(* CODESYS project Flight Simulator.project
   CompiledLibraryCompatibilityVersion: CODESYS V3.5 SP16 Patch 7

Project tree, tasks and I/O mapping:
  PLC : HX-CP1S08, Hitachi Industrial Equipment Systems Co., Ltd., order no. HX-CP1S08, version 3.5.8.24
      settings: IP Address = '192.168.137.20'
    application Application
      libraries: Unit Conversion Interfaces, * (Intern); Standard, * (System); VisuDialogs, * (System); CAA Device Diagnosis, 3.5.4.0 (CAA Technical Workgroup); CAA Net Base Services, 3.5.8.10 (CAA Technical Workgroup); NetVarUdp, 3.5.17.0 (System); PRO JSON, 1.0.0.13 (Pro Electric)
      task EtherCAT_Task (cyclic, interval 8 ms, priority 1) calls nothing
      task VISU_TASK (cyclic, interval 200 ms, priority 31) calls VisuElems.Visu_Prg
      task Task (cyclic, interval 5 ms, priority 1) calls main, TcpClient
      global variables gvlSetting
      data type ServoData
      program TcpClient [ST]
      program main [ST]
      visualisation Main
      global variables GVL
    SoftMotion General Axis Pool : SoftMotion General Axis Pool, 3S - Smart Software Solutions GmbH, version 4.9.0.0
      SM_Drive_Virtual : SM_Drive_Virtual, 3S - Smart Software Solutions GmbH, order no. 1805, version 4.0.0.0
          settings: wDriveID = 6
    Basic : Basic, Hitachi-IES, version 3.5.8.20
      _16_Digital_Input : 16 Digital Input, Hitachi-IES, version 3.4.0.0
          input  Application.GVL.resetButton : BOOL  // ReserveWord0Type.Bit1
          input  Application.GVL.startButton : BOOL  // ReserveWord0Type.Bit2
          input  Application.GVL.stopButton : BOOL  // ReserveWord0Type.Bit3
          input  Application.GVL.safetySystem : BOOL  // ReserveWord0Type.Bit4
          unmapped channels: ReserveWord0Type, ReserveWord0Type, ReserveWord0Type
      _16_Digital_Output : 16 Digital Output, Hitachi-IES, version 3.4.0.0
          output Application.GVL.LightGreen : BOOL  // ReserveWord0Type.Bit0
          output Application.GVL.LightYellow : BOOL  // ReserveWord0Type.Bit1
          output Application.GVL.LightRed : BOOL  // ReserveWord0Type.Bit2
          unmapped channels: ReserveWord0Type, ReserveWord0Type, ReserveWord0Type
      <Empty>
      <Empty>
      _16_Digital_Input_1 : 16 Digital Input, Hitachi-IES, version 3.4.0.0
          unmapped channels: ReserveWord0Type, ReserveWord0Type, ReserveWord0Type
      <Empty>
      <Empty>
      <Empty>
      <Empty>
      <Empty>
      _16_Digital_Output_1 : 16 Digital Output, Hitachi-IES, version 3.4.0.0
          unmapped channels: ReserveWord0Type, ReserveWord0Type, ReserveWord0Type
    EtherCAT_Master : EtherCAT Master, Festo, version 3.5.16.43
        settings: MasterUseLRW = False; SlaveAutoRestart = True; NetworkName = 'eth2'; NetworkName = "eth2"; SelectNetworkByName = False; EnableTaskMessage = False; SrcAddress1 = 42135; SrcAddress2 = 3137775364; EnableSecondAdapter = False; SrcAddress = [16#A4,16#97,16#BB,16#06,16#A7,16#04]; NetworkName = 'eth2'; NetworkName = "eth2"; SelectNetworkByName = False
      servo_drive_2 : CMMT-AS (SoftMotion), Festo, order no. 5340819, 5340820, version 4.0.20.0
          settings: StationAlias = 0; Number of SDO = 1; Modes of operation.Index = 16#6060; Modes of operation.Subindex = 16#00; Modes of operation.Value = 8; Modes of operation.Size = 8; Modes of operation.AbortIfError = FALSE; Modes of operation.JumpToLine = FALSE; Modes of operation.Line = 0; Modes of operation.CompleteAccess = False
          unmapped channels: Controlword, Modes of operation, Target position, Profile velocity, Target velocity, Target torque, Velocity offset, Torque offset, Touch probe function, ---, Statusword, Modes of operation display, Position actual value, Velocity actual value, Torque actual value, Touch probe status, Touch probe 1 positive edge, Touch probe 1 negative edge, Touch probe 2 positive edge, Touch probe 2 negative edge, ---
        SM_Drive_EtherCAT_Festo_CMMT_AS_1 : SM_Drive_EtherCAT_Festo_CMMT_AS, Festo, version 4.0.20.0
            settings: AdrOffset_8010 = 36; BitOffset_8010 = 0; BitLength_8010 = 16; Address_8010 = '%QW18'; Type_8010 = 'UINT'; AddressPointer_8010 = ADR(%QW18); AdrOffset_8020 = 38; BitOffset_8020 = 0; BitLength_8020 = 8; Address_8020 = '%QB38'; Type_8020 = 'SINT'; AddressPointer_8020 = ADR(%QB38); AdrOffset_8030 = 40; BitOffset_8030 = 0; BitLength_8030 = 32; Address_8030 = '%QD10'; Type_8030 = 'DINT'; AddressPointer_8030 = ADR(%QD10); AdrOffset_8040 = 48; BitOffset_8040 = 0; BitLength_8040 = 32; Address_8040 = '%QD12'; Type_8040 = 'DINT'; AddressPointer_8040 = ADR(%QD12); AdrOffset_8050 = 52; BitOffset_8050 = 0; BitLength_8050 = 16; Address_8050 = '%QW26'; Type_8050 = 'INT'; AddressPointer_8050 = ADR(%QW26); AdrOffset_8060 = 62; BitOffset_8060 = 0; BitLength_8060 = 16; Address_8060 = '%QW31'; Type_8060 = 'UINT'; AddressPointer_8060 = ADR(%QW31); AdrOffset_8510 = 40; BitOffset_8510 = 0; BitLength_8510 = 16; Address_8510 = '%IW20';
              Type_8510 = 'UINT'; AddressPointer_8510 = ADR(%IW20); AdrOffset_8520 = 42; BitOffset_8520 = 0; BitLength_8520 = 8; Address_8520 = '%IB42'; Type_8520 = 'SINT'; AddressPointer_8520 = ADR(%IB42); AdrOffset_8530 = 44; BitOffset_8530 = 0; BitLength_8530 = 32; Address_8530 = '%ID11'; Type_8530 = 'DINT'; AddressPointer_8530 = ADR(%ID11); AdrOffset_8540 = 48; BitOffset_8540 = 0; BitLength_8540 = 32; Address_8540 = '%ID12'; Type_8540 = 'DINT'; AddressPointer_8540 = ADR(%ID12); AdrOffset_8550 = 52; BitOffset_8550 = 0; BitLength_8550 = 16; Address_8550 = '%IW26'; Type_8550 = 'INT'; AddressPointer_8550 = ADR(%IW26); AdrOffset_8560 = 54; BitOffset_8560 = 0; BitLength_8560 = 16; Address_8560 = '%IW27'; Type_8560 = 'UINT'; AddressPointer_8560 = ADR(%IW27); AdrOffset_8570 = 56; BitOffset_8570 = 0; BitLength_8570 = 32; Address_8570 = '%ID14'; Type_8570 = 'DINT'; AddressPointer_8570 = ADR(%ID14); AdrOffset_8580 = 60; BitOffset_8580 = 0;
              BitLength_8580 = 32; Address_8580 = '%ID15'; Type_8580 = 'DINT'; AddressPointer_8580 = ADR(%ID15); AdrOffset_8590 = 64; BitOffset_8590 = 0; BitLength_8590 = 32; Address_8590 = '%ID16'; Type_8590 = 'DINT'; AddressPointer_8590 = ADR(%ID16); AdrOffset_8600 = 68; BitOffset_8600 = 0; BitLength_8600 = 32; Address_8600 = '%ID17'; Type_8600 = 'DINT'; AddressPointer_8600 = ADR(%ID17)
      servo_drive_1 : CMMT-AS (SoftMotion), Festo, order no. 5340819, 5340820, version 4.0.20.0
          settings: StationAlias = 0; Number of SDO = 1; Modes of operation.Index = 16#6060; Modes of operation.Subindex = 16#00; Modes of operation.Value = 8; Modes of operation.Size = 8; Modes of operation.AbortIfError = FALSE; Modes of operation.JumpToLine = FALSE; Modes of operation.Line = 0; Modes of operation.CompleteAccess = False
          unmapped channels: Controlword, Modes of operation, Target position, Profile velocity, Target velocity, Target torque, Velocity offset, Torque offset, Touch probe function, ---, Statusword, Modes of operation display, Position actual value, Velocity actual value, Torque actual value, Touch probe status, Touch probe 1 positive edge, Touch probe 1 negative edge, Touch probe 2 positive edge, Touch probe 2 negative edge, ---
        SM_Drive_EtherCAT_Festo_CMMT_AS : SM_Drive_EtherCAT_Festo_CMMT_AS, Festo, version 4.0.20.0
            settings: wDriveID = 0; AdrOffset_8010 = 4; BitOffset_8010 = 0; BitLength_8010 = 16; Address_8010 = '%QW2'; Type_8010 = 'UINT'; AddressPointer_8010 = ADR(%QW2); AdrOffset_8020 = 6; BitOffset_8020 = 0; BitLength_8020 = 8; Address_8020 = '%QB6'; Type_8020 = 'SINT'; AddressPointer_8020 = ADR(%QB6); AdrOffset_8030 = 8; BitOffset_8030 = 0; BitLength_8030 = 32; Address_8030 = '%QD2'; Type_8030 = 'DINT'; AddressPointer_8030 = ADR(%QD2); AdrOffset_8040 = 16; BitOffset_8040 = 0; BitLength_8040 = 32; Address_8040 = '%QD4'; Type_8040 = 'DINT'; AddressPointer_8040 = ADR(%QD4); AdrOffset_8050 = 20; BitOffset_8050 = 0; BitLength_8050 = 16; Address_8050 = '%QW10'; Type_8050 = 'INT'; AddressPointer_8050 = ADR(%QW10); AdrOffset_8060 = 30; BitOffset_8060 = 0; BitLength_8060 = 16; Address_8060 = '%QW15'; Type_8060 = 'UINT'; AddressPointer_8060 = ADR(%QW15); AdrOffset_8510 = 4; BitOffset_8510 = 0; BitLength_8510 = 16;
              Address_8510 = '%IW2'; Type_8510 = 'UINT'; AddressPointer_8510 = ADR(%IW2); AdrOffset_8520 = 6; BitOffset_8520 = 0; BitLength_8520 = 8; Address_8520 = '%IB6'; Type_8520 = 'SINT'; AddressPointer_8520 = ADR(%IB6); AdrOffset_8530 = 8; BitOffset_8530 = 0; BitLength_8530 = 32; Address_8530 = '%ID2'; Type_8530 = 'DINT'; AddressPointer_8530 = ADR(%ID2); AdrOffset_8540 = 12; BitOffset_8540 = 0; BitLength_8540 = 32; Address_8540 = '%ID3'; Type_8540 = 'DINT'; AddressPointer_8540 = ADR(%ID3); AdrOffset_8550 = 16; BitOffset_8550 = 0; BitLength_8550 = 16; Address_8550 = '%IW8'; Type_8550 = 'INT'; AddressPointer_8550 = ADR(%IW8); AdrOffset_8560 = 18; BitOffset_8560 = 0; BitLength_8560 = 16; Address_8560 = '%IW9'; Type_8560 = 'UINT'; AddressPointer_8560 = ADR(%IW9); AdrOffset_8570 = 20; BitOffset_8570 = 0; BitLength_8570 = 32; Address_8570 = '%ID5'; Type_8570 = 'DINT'; AddressPointer_8570 = ADR(%ID5); AdrOffset_8580 = 24;
              BitOffset_8580 = 0; BitLength_8580 = 32; Address_8580 = '%ID6'; Type_8580 = 'DINT'; AddressPointer_8580 = ADR(%ID6); AdrOffset_8590 = 28; BitOffset_8590 = 0; BitLength_8590 = 32; Address_8590 = '%ID7'; Type_8590 = 'DINT'; AddressPointer_8590 = ADR(%ID7); AdrOffset_8600 = 32; BitOffset_8600 = 0; BitLength_8600 = 32; Address_8600 = '%ID8'; Type_8600 = 'DINT'; AddressPointer_8600 = ADR(%ID8)
      servo_drive_3 : CMMT-AS (SoftMotion), Festo, order no. 5340819, 5340820, version 4.0.22.0
          settings: StationAlias = 0; Number of SDO = 1; Modes of operation.Index = 16#6060; Modes of operation.Subindex = 16#00; Modes of operation.Value = 8; Modes of operation.Size = 8; Modes of operation.AbortIfError = FALSE; Modes of operation.JumpToLine = FALSE; Modes of operation.Line = 0; Modes of operation.CompleteAccess = False
          unmapped channels: Controlword, Modes of operation, Target position, Profile velocity, Target velocity, Target torque, Velocity offset, Torque offset, Touch probe function, ---, Statusword, Modes of operation display, Position actual value, Velocity actual value, Torque actual value, Touch probe status, Touch probe 1 positive edge, Touch probe 1 negative edge, Touch probe 2 positive edge, Touch probe 2 negative edge, ---
        SM_Drive_EtherCAT_Festo_CMMT_AS_2 : SM_Drive_EtherCAT_Festo_CMMT_AS, Festo, version 4.0.22.0
            settings: wDriveID = 2; AdrOffset_8010 = 68; BitOffset_8010 = 0; BitLength_8010 = 16; Address_8010 = '%QW34'; Type_8010 = 'UINT'; AddressPointer_8010 = ADR(%QW34); AdrOffset_8020 = 70; BitOffset_8020 = 0; BitLength_8020 = 8; Address_8020 = '%QB70'; Type_8020 = 'SINT'; AddressPointer_8020 = ADR(%QB70); AdrOffset_8030 = 72; BitOffset_8030 = 0; BitLength_8030 = 32; Address_8030 = '%QD18'; Type_8030 = 'DINT'; AddressPointer_8030 = ADR(%QD18); AdrOffset_8040 = 80; BitOffset_8040 = 0; BitLength_8040 = 32; Address_8040 = '%QD20'; Type_8040 = 'DINT'; AddressPointer_8040 = ADR(%QD20); AdrOffset_8050 = 84; BitOffset_8050 = 0; BitLength_8050 = 16; Address_8050 = '%QW42'; Type_8050 = 'INT'; AddressPointer_8050 = ADR(%QW42); AdrOffset_8060 = 94; BitOffset_8060 = 0; BitLength_8060 = 16; Address_8060 = '%QW47'; Type_8060 = 'UINT'; AddressPointer_8060 = ADR(%QW47); AdrOffset_8510 = 76; BitOffset_8510 = 0; BitLength_8510 = 16;
              Address_8510 = '%IW38'; Type_8510 = 'UINT'; AddressPointer_8510 = ADR(%IW38); AdrOffset_8520 = 78; BitOffset_8520 = 0; BitLength_8520 = 8; Address_8520 = '%IB78'; Type_8520 = 'SINT'; AddressPointer_8520 = ADR(%IB78); AdrOffset_8530 = 80; BitOffset_8530 = 0; BitLength_8530 = 32; Address_8530 = '%ID20'; Type_8530 = 'DINT'; AddressPointer_8530 = ADR(%ID20); AdrOffset_8540 = 84; BitOffset_8540 = 0; BitLength_8540 = 32; Address_8540 = '%ID21'; Type_8540 = 'DINT'; AddressPointer_8540 = ADR(%ID21); AdrOffset_8550 = 88; BitOffset_8550 = 0; BitLength_8550 = 16; Address_8550 = '%IW44'; Type_8550 = 'INT'; AddressPointer_8550 = ADR(%IW44); AdrOffset_8560 = 90; BitOffset_8560 = 0; BitLength_8560 = 16; Address_8560 = '%IW45'; Type_8560 = 'UINT'; AddressPointer_8560 = ADR(%IW45); AdrOffset_8570 = 92; BitOffset_8570 = 0; BitLength_8570 = 32; Address_8570 = '%ID23'; Type_8570 = 'DINT'; AddressPointer_8570 = ADR(%ID23); AdrOffset_8580 = 96;
              BitOffset_8580 = 0; BitLength_8580 = 32; Address_8580 = '%ID24'; Type_8580 = 'DINT'; AddressPointer_8580 = ADR(%ID24); AdrOffset_8590 = 100; BitOffset_8590 = 0; BitLength_8590 = 32; Address_8590 = '%ID25'; Type_8590 = 'DINT'; AddressPointer_8590 = ADR(%ID25); AdrOffset_8600 = 104; BitOffset_8600 = 0; BitLength_8600 = 32; Address_8600 = '%ID26'; Type_8600 = 'DINT'; AddressPointer_8600 = ADR(%ID26)
      servo_drive_4 : CMMT-AS (SoftMotion), Festo, order no. 5340819, 5340820, version 4.0.20.0
          settings: StationAlias = 0; Number of SDO = 1; Modes of operation.Index = 16#6060; Modes of operation.Subindex = 16#00; Modes of operation.Value = 8; Modes of operation.Size = 8; Modes of operation.AbortIfError = FALSE; Modes of operation.JumpToLine = FALSE; Modes of operation.Line = 0; Modes of operation.CompleteAccess = False
          unmapped channels: Controlword, Modes of operation, Target position, Profile velocity, Target velocity, Target torque, Velocity offset, Torque offset, Touch probe function, ---, Statusword, Modes of operation display, Position actual value, Velocity actual value, Torque actual value, Touch probe status, Touch probe 1 positive edge, Touch probe 1 negative edge, Touch probe 2 positive edge, Touch probe 2 negative edge, ---
        SM_Drive_EtherCAT_Festo_CMMT_AS_3 : SM_Drive_EtherCAT_Festo_CMMT_AS, Festo, version 4.0.20.0
            settings: wDriveID = 3; AdrOffset_8010 = 100; BitOffset_8010 = 0; BitLength_8010 = 16; Address_8010 = '%QW50'; Type_8010 = 'UINT'; AddressPointer_8010 = ADR(%QW50); AdrOffset_8020 = 102; BitOffset_8020 = 0; BitLength_8020 = 8; Address_8020 = '%QB102'; Type_8020 = 'SINT'; AddressPointer_8020 = ADR(%QB102); AdrOffset_8030 = 104; BitOffset_8030 = 0; BitLength_8030 = 32; Address_8030 = '%QD26'; Type_8030 = 'DINT'; AddressPointer_8030 = ADR(%QD26); AdrOffset_8040 = 112; BitOffset_8040 = 0; BitLength_8040 = 32; Address_8040 = '%QD28'; Type_8040 = 'DINT'; AddressPointer_8040 = ADR(%QD28); AdrOffset_8050 = 116; BitOffset_8050 = 0; BitLength_8050 = 16; Address_8050 = '%QW58'; Type_8050 = 'INT'; AddressPointer_8050 = ADR(%QW58); AdrOffset_8060 = 126; BitOffset_8060 = 0; BitLength_8060 = 16; Address_8060 = '%QW63'; Type_8060 = 'UINT'; AddressPointer_8060 = ADR(%QW63); AdrOffset_8510 = 112; BitOffset_8510 = 0; BitLength_8510 = 16;
              Address_8510 = '%IW56'; Type_8510 = 'UINT'; AddressPointer_8510 = ADR(%IW56); AdrOffset_8520 = 114; BitOffset_8520 = 0; BitLength_8520 = 8; Address_8520 = '%IB114'; Type_8520 = 'SINT'; AddressPointer_8520 = ADR(%IB114); AdrOffset_8530 = 116; BitOffset_8530 = 0; BitLength_8530 = 32; Address_8530 = '%ID29'; Type_8530 = 'DINT'; AddressPointer_8530 = ADR(%ID29); AdrOffset_8540 = 120; BitOffset_8540 = 0; BitLength_8540 = 32; Address_8540 = '%ID30'; Type_8540 = 'DINT'; AddressPointer_8540 = ADR(%ID30); AdrOffset_8550 = 124; BitOffset_8550 = 0; BitLength_8550 = 16; Address_8550 = '%IW62'; Type_8550 = 'INT'; AddressPointer_8550 = ADR(%IW62); AdrOffset_8560 = 126; BitOffset_8560 = 0; BitLength_8560 = 16; Address_8560 = '%IW63'; Type_8560 = 'UINT'; AddressPointer_8560 = ADR(%IW63); AdrOffset_8570 = 128; BitOffset_8570 = 0; BitLength_8570 = 32; Address_8570 = '%ID32'; Type_8570 = 'DINT'; AddressPointer_8570 = ADR(%ID32); AdrOffset_8580 = 132;
              BitOffset_8580 = 0; BitLength_8580 = 32; Address_8580 = '%ID33'; Type_8580 = 'DINT'; AddressPointer_8580 = ADR(%ID33); AdrOffset_8590 = 136; BitOffset_8590 = 0; BitLength_8590 = 32; Address_8590 = '%ID34'; Type_8590 = 'DINT'; AddressPointer_8590 = ADR(%ID34); AdrOffset_8600 = 140; BitOffset_8600 = 0; BitLength_8600 = 32; Address_8600 = '%ID35'; Type_8600 = 'DINT'; AddressPointer_8600 = ADR(%ID35)
      servo_drive_5 : CMMT-AS (SoftMotion), Festo, order no. 5340819, 5340820, version 4.0.20.0
          settings: StationAlias = 0; Number of SDO = 1; Modes of operation.Index = 16#6060; Modes of operation.Subindex = 16#00; Modes of operation.Value = 8; Modes of operation.Size = 8; Modes of operation.AbortIfError = FALSE; Modes of operation.JumpToLine = FALSE; Modes of operation.Line = 0; Modes of operation.CompleteAccess = False
          unmapped channels: Controlword, Modes of operation, Target position, Profile velocity, Target velocity, Target torque, Velocity offset, Torque offset, Touch probe function, ---, Statusword, Modes of operation display, Position actual value, Velocity actual value, Torque actual value, Touch probe status, Touch probe 1 positive edge, Touch probe 1 negative edge, Touch probe 2 positive edge, Touch probe 2 negative edge, ---
        SM_Drive_EtherCAT_Festo_CMMT_AS_4 : SM_Drive_EtherCAT_Festo_CMMT_AS, Festo, version 4.0.20.0
            settings: wDriveID = 4; AdrOffset_8010 = 132; BitOffset_8010 = 0; BitLength_8010 = 16; Address_8010 = '%QW66'; Type_8010 = 'UINT'; AddressPointer_8010 = ADR(%QW66); AdrOffset_8020 = 134; BitOffset_8020 = 0; BitLength_8020 = 8; Address_8020 = '%QB134'; Type_8020 = 'SINT'; AddressPointer_8020 = ADR(%QB134); AdrOffset_8030 = 136; BitOffset_8030 = 0; BitLength_8030 = 32; Address_8030 = '%QD34'; Type_8030 = 'DINT'; AddressPointer_8030 = ADR(%QD34); AdrOffset_8040 = 144; BitOffset_8040 = 0; BitLength_8040 = 32; Address_8040 = '%QD36'; Type_8040 = 'DINT'; AddressPointer_8040 = ADR(%QD36); AdrOffset_8050 = 148; BitOffset_8050 = 0; BitLength_8050 = 16; Address_8050 = '%QW74'; Type_8050 = 'INT'; AddressPointer_8050 = ADR(%QW74); AdrOffset_8060 = 158; BitOffset_8060 = 0; BitLength_8060 = 16; Address_8060 = '%QW79'; Type_8060 = 'UINT'; AddressPointer_8060 = ADR(%QW79); AdrOffset_8510 = 148; BitOffset_8510 = 0; BitLength_8510 = 16;
              Address_8510 = '%IW74'; Type_8510 = 'UINT'; AddressPointer_8510 = ADR(%IW74); AdrOffset_8520 = 150; BitOffset_8520 = 0; BitLength_8520 = 8; Address_8520 = '%IB150'; Type_8520 = 'SINT'; AddressPointer_8520 = ADR(%IB150); AdrOffset_8530 = 152; BitOffset_8530 = 0; BitLength_8530 = 32; Address_8530 = '%ID38'; Type_8530 = 'DINT'; AddressPointer_8530 = ADR(%ID38); AdrOffset_8540 = 156; BitOffset_8540 = 0; BitLength_8540 = 32; Address_8540 = '%ID39'; Type_8540 = 'DINT'; AddressPointer_8540 = ADR(%ID39); AdrOffset_8550 = 160; BitOffset_8550 = 0; BitLength_8550 = 16; Address_8550 = '%IW80'; Type_8550 = 'INT'; AddressPointer_8550 = ADR(%IW80); AdrOffset_8560 = 162; BitOffset_8560 = 0; BitLength_8560 = 16; Address_8560 = '%IW81'; Type_8560 = 'UINT'; AddressPointer_8560 = ADR(%IW81); AdrOffset_8570 = 164; BitOffset_8570 = 0; BitLength_8570 = 32; Address_8570 = '%ID41'; Type_8570 = 'DINT'; AddressPointer_8570 = ADR(%ID41); AdrOffset_8580 = 168;
              BitOffset_8580 = 0; BitLength_8580 = 32; Address_8580 = '%ID42'; Type_8580 = 'DINT'; AddressPointer_8580 = ADR(%ID42); AdrOffset_8590 = 172; BitOffset_8590 = 0; BitLength_8590 = 32; Address_8590 = '%ID43'; Type_8590 = 'DINT'; AddressPointer_8590 = ADR(%ID43); AdrOffset_8600 = 176; BitOffset_8600 = 0; BitLength_8600 = 32; Address_8600 = '%ID44'; Type_8600 = 'DINT'; AddressPointer_8600 = ADR(%ID44)
      servo_drive_6 : CMMT-AS (SoftMotion), Festo, order no. 5340819, 5340820, version 4.0.20.0
          settings: StationAlias = 0; Number of SDO = 1; Modes of operation.Index = 16#6060; Modes of operation.Subindex = 16#00; Modes of operation.Value = 8; Modes of operation.Size = 8; Modes of operation.AbortIfError = FALSE; Modes of operation.JumpToLine = FALSE; Modes of operation.Line = 0; Modes of operation.CompleteAccess = False
          unmapped channels: Controlword, Modes of operation, Target position, Profile velocity, Target velocity, Target torque, Velocity offset, Torque offset, Touch probe function, ---, Statusword, Modes of operation display, Position actual value, Velocity actual value, Torque actual value, Touch probe status, Touch probe 1 positive edge, Touch probe 1 negative edge, Touch probe 2 positive edge, Touch probe 2 negative edge, ---
        SM_Drive_EtherCAT_Festo_CMMT_AS_5 : SM_Drive_EtherCAT_Festo_CMMT_AS, Festo, version 4.0.20.0
            settings: wDriveID = 5; AdrOffset_8010 = 164; BitOffset_8010 = 0; BitLength_8010 = 16; Address_8010 = '%QW82'; Type_8010 = 'UINT'; AddressPointer_8010 = ADR(%QW82); AdrOffset_8020 = 166; BitOffset_8020 = 0; BitLength_8020 = 8; Address_8020 = '%QB166'; Type_8020 = 'SINT'; AddressPointer_8020 = ADR(%QB166); AdrOffset_8030 = 168; BitOffset_8030 = 0; BitLength_8030 = 32; Address_8030 = '%QD42'; Type_8030 = 'DINT'; AddressPointer_8030 = ADR(%QD42); AdrOffset_8040 = 176; BitOffset_8040 = 0; BitLength_8040 = 32; Address_8040 = '%QD44'; Type_8040 = 'DINT'; AddressPointer_8040 = ADR(%QD44); AdrOffset_8050 = 180; BitOffset_8050 = 0; BitLength_8050 = 16; Address_8050 = '%QW90'; Type_8050 = 'INT'; AddressPointer_8050 = ADR(%QW90); AdrOffset_8060 = 190; BitOffset_8060 = 0; BitLength_8060 = 16; Address_8060 = '%QW95'; Type_8060 = 'UINT'; AddressPointer_8060 = ADR(%QW95); AdrOffset_8510 = 184; BitOffset_8510 = 0; BitLength_8510 = 16;
              Address_8510 = '%IW92'; Type_8510 = 'UINT'; AddressPointer_8510 = ADR(%IW92); AdrOffset_8520 = 186; BitOffset_8520 = 0; BitLength_8520 = 8; Address_8520 = '%IB186'; Type_8520 = 'SINT'; AddressPointer_8520 = ADR(%IB186); AdrOffset_8530 = 188; BitOffset_8530 = 0; BitLength_8530 = 32; Address_8530 = '%ID47'; Type_8530 = 'DINT'; AddressPointer_8530 = ADR(%ID47); AdrOffset_8540 = 192; BitOffset_8540 = 0; BitLength_8540 = 32; Address_8540 = '%ID48'; Type_8540 = 'DINT'; AddressPointer_8540 = ADR(%ID48); AdrOffset_8550 = 196; BitOffset_8550 = 0; BitLength_8550 = 16; Address_8550 = '%IW98'; Type_8550 = 'INT'; AddressPointer_8550 = ADR(%IW98); AdrOffset_8560 = 198; BitOffset_8560 = 0; BitLength_8560 = 16; Address_8560 = '%IW99'; Type_8560 = 'UINT'; AddressPointer_8560 = ADR(%IW99); AdrOffset_8570 = 200; BitOffset_8570 = 0; BitLength_8570 = 32; Address_8570 = '%ID50'; Type_8570 = 'DINT'; AddressPointer_8570 = ADR(%ID50); AdrOffset_8580 = 204;
              BitOffset_8580 = 0; BitLength_8580 = 32; Address_8580 = '%ID51'; Type_8580 = 'DINT'; AddressPointer_8580 = ADR(%ID51); AdrOffset_8590 = 208; BitOffset_8590 = 0; BitLength_8590 = 32; Address_8590 = '%ID52'; Type_8590 = 'DINT'; AddressPointer_8590 = ADR(%ID52); AdrOffset_8600 = 212; BitOffset_8600 = 0; BitLength_8600 = 32; Address_8600 = '%ID53'; Type_8600 = 'DINT'; AddressPointer_8600 = ADR(%ID53)
  libraries: VisuSymbols, 4.1.0.0 (System)
  function block Axis [ST]: enabled, init, doAbort, isReady, doMovement, doReset, getPosition, inError, cycle, isInitialised
  function block signal [ST]: init, cycle
  text list GlobalTextList
  function block Light [ST]: blink, init, cycle, enable
  function block FlightSimulator [ST]: safetyStop, doReset, isEnabled, getPositions, cycle, goNeutralPosition, isReady, doMovement, isInitialised, init, inError, goHomePosition, goTopPosition
  data type stateFlightSimulator
*)

// PLC/Application/ServoData
TYPE ServoData :
STRUCT
	positions: ARRAY[1..6] OF JSONVAR;
	speeds: ARRAY[1..6] OF JSONVAR;
END_STRUCT
END_TYPE

// stateFlightSimulator
{attribute 'qualified_only'}
{attribute 'strict'}
TYPE stateFlightSimulator :
(
	error  := 0,
	resetting,
	stopped,
	starting,
	started,
	stopping
);
END_TYPE

// PLC/Application/gvlSetting
{attribute 'qualified_only'}
VAR_GLOBAL CONSTANT
    // Port to use to send data.
	gc_uiPort        : UINT := 32760;
    // IP Address of the computer that hosts the software.
	gc_stIpAddr      : NBS.IP_ADDR := (sAddr := '192.168.137.123');
	// Length of the telegram.
    gc_wMaxTelegram  : INT := 512;
END_VAR

// PLC/Application/GVL
{attribute 'qualified_only'}
VAR_GLOBAL
	// Red light on electrical housing.
	lightRed: BOOL;
	// Yellow light on electrical housing.
	lightYellow: BOOL;
	// Green light on electrical housing.
	lightGreen: BOOL;
	// Reset button on electrical housing.
	resetButton: BOOL := FALSE;
	// Start button on electrical housing.
	startButton: BOOL := FALSE;
	// Stop button on electrical housing.
	stopButton: BOOL := FALSE;
	// Safety system, connected to safety relay.
	safetySystem: BOOL := FALSE;
	// Virtual reset button on HMI.
	resetHMI: BOOL;
	// Virtual start button on HMI.
	startHMI: BOOL;
	// Virtual stop button on HMI.
	stopHMI: BOOL;
	// Virtual toggle button to toggle between tCP data and manual data on HMI.
	useTCPData: BOOL := TRUE;
	// Manual slider velocity input on HMI.
	nextVelocityInput: REAL := 200;
	// Manual slider position input on HMI.
	nextPositionInput: REAL := 0;
	// Flight simulator object.
	FlightSimulator: FlightSimulator;
	// Velocity input from TCP data or HMI data.
	servoVelocities: ARRAY[1..6] OF REAL;
	// Position input from TCP data or HMI data.
	servoPositions: ARRAY[1..6] OF REAL;
	// Current Positions in array format.
	servoPositionsCurrent: ARRAY[1..6] OF REAL;
	// Current Positions in JSON format, used to send back to TCP client.
	currentPositions: ARRAY[1..6] OF JSONVAR;
END_VAR

// PLC/Application/main
PROGRAM main
VAR
	bInit: BOOL := TRUE;
	iCounter : INT;
	bEnabled: BOOL;
	iDataUpdated: INT := 0;
	tonTimer: TON;
	UpdateCount: INT := 0;
END_VAR

IF bInit THEN
	GVL.FlightSimulator.init(
		axis1 := SM_Drive_EtherCAT_Festo_CMMT_AS,
		axis2 := SM_Drive_EtherCAT_Festo_CMMT_AS_1,
		axis3 := SM_Drive_EtherCAT_Festo_CMMT_AS_2,
		axis4 := SM_Drive_EtherCAT_Festo_CMMT_AS_3,
		axis5 := SM_Drive_EtherCAT_Festo_CMMT_AS_4,
		axis6 := SM_Drive_EtherCAT_Festo_CMMT_AS_5,
		GVL.lightRed,
		GVL.lightYellow,
		GVL.lightGreen,
		enabled := bEnabled,
		safetySystem := GVL.safetySystem,
		newPositions := GVL.servoPositions,
		newVelocities := GVL.servoVelocities
	);
	bInit := FALSE;
END_IF

// Handle reset buttons.
IF GVL.resetButton OR GVL.resetHMI THEN // blauwe knop
	bEnabled := FALSE;
	GVL.FlightSimulator.doReset();
	
	// [NEW] Reset position data zodat platform niet naar oude waarden springt
	FOR iCounter := 1 TO 6 DO
		GVL.currentPositions[iCounter].Number := 0.0;
		GVL.servoPositions[iCounter] := 0.0;
		GVL.servoVelocities[iCounter] := 0.0;
	END_FOR
END_IF

// Handle start buttons.
IF GVL.startButton OR GVL.startHMI THEN // witte knop
	bEnabled := TRUE;
END_IF

// Handle stop buttons
IF GVL.stopButton OR GVL.stopHMI THEN // zwarte knop
	bEnabled := FALSE;
END_IF

// Go through all positions and velocities.
FOR iCounter := 1 TO 6 BY 1 DO 
	IF GVL.useTCPData THEN
		// Always use latest TCP data (don't wait for parseJSON.Done)
		GVL.servoPositions[iCounter] := tcpClient.servoData.positions[iCounter].Number;
		GVL.servoVelocities[iCounter] := tcpClient.servoData.speeds[iCounter].Number;
		
		// Optional: track successful updates for diagnostics
		IF tcpClient.parseJSON.Done THEN
			UpdateCount := UpdateCount + 1;
		END_IF
	ELSE
		// Else take the data from the sliders from the HMI.
		GVL.servoPositions[iCounter] := GVL.nextPositionInput;
		GVL.servoVelocities[iCounter] := GVL.nextVelocityInput;
	END_IF
END_FOR

//THIS^.signal.green.enable := FALSE;
//THIS^.signal.green.blink := FALSE;
//THIS^.signal.green.enable := FALSE;
//THIS^.signal.green.blink := FALSE;

// Cycle sub functions.
GVL.FlightSimulator.cycle();

// Get current positions, used for TcpClient.
FOR iCounter := 1 TO 6 BY 1 DO
	GVL.currentPositions[iCounter].Number := GVL.FlightSimulator.axis[iCounter].getPosition();
	GVL.servoPositionsCurrent[iCounter] := GVL.FlightSimulator.axis[iCounter].getPosition();
END_FOR

END_PROGRAM

// FlightSimulator
FUNCTION_BLOCK FlightSimulator
VAR_OUTPUT
	// Axis objects.
	axis: ARRAY[1..6] OF Axis;
	// Signal objects.
	signal: signal;
END_VAR
VAR
	// Current state of flight simulator.
	state: stateFlightSimulator;
	// Used in some states to add extra delay.
	bToggle: BOOL;
	// REF to if system should be enabled.
	enabled: REFERENCE TO BOOL;
	// REF to safety system.
	safetySystem: REFERENCE TO BOOL;
	// REF to new positions.
	newPositions: REFERENCE TO ARRAY[1..6] OF REAL;
	// REF to new velocities.
	newVelocities: REFERENCE TO ARRAY[1..6] OF REAL;
END_VAR

METHOD safetyStop : BOOL
VAR
	// Counter to cycle through axis.
	iCounter: UINT;
END_VAR
// Disable all axis.
FOR iCounter := 1 TO 6 BY 1 DO
	THIS^.axis[iCounter].enabled := FALSE;
END_FOR
THIS^.enabled := FALSE;
END_METHOD

METHOD doReset : BOOL
VAR_INPUT
END_VAR
VAR
	// Counter to cycle through axis.
	iCounter: UINT;
END_VAR
THIS^.state := stateFlightSimulator.resetting;
END_METHOD

METHOD isEnabled : BOOL;
VAR_INPUT
END_VAR
VAR
	// Counter to cycle through axis.
	iCounter: INT;
END_VAR
// Check enabled status of all axis, when one is not enabled return with FALSE.
FOR iCounter := 1 TO 6 BY 1 DO
	IF NOT THIS^.axis[iCounter].enabled THEN
		isEnabled := FALSE;
		RETURN;
	END_IF;
END_FOR;

isEnabled := TRUE;
END_METHOD

METHOD getPositions : ARRAY[1..6] OF REAL
VAR_INPUT
END_VAR
VAR
	// Counter to cycle through axis.
	iCounter: INT;
END_VAR
// Write current axis positions
FOR iCounter := 1 TO 6 BY 1 DO
	getPositions[iCounter] := THIS^.axis[iCounter].getPosition();
END_FOR
END_METHOD

METHOD cycle : BOOL
VAR
	// Counter to cycle through axis.
	iCounter: UINT;
END_VAR
// If safety system has been triggered/broken go to error.
IF NOT THIS^.safetySystem THEN
	THIS^.state := stateFlightSimulator.error;
	THIS^.safetyStop();
END_IF

// If any Axis is in error stop all axis.
IF THIS^.inError() AND NOT (THIS^.state = stateFlightSimulator.error) THEN
	IF NOT (THIS^.state = stateFlightSimulator.resetting) THEN
		THIS^.state := stateFlightSimulator.error;
		THIS^.safetyStop();
	END_IF
END_IF

// Reset signal variables.
THIS^.signal.red.enable := FALSE;
THIS^.signal.yellow.enable := FALSE;
THIS^.signal.green.enable := FALSE;
THIS^.signal.red.blink := FALSE;
THIS^.signal.yellow.blink := FALSE;
THIS^.signal.green.blink := FALSE;

// Status case switch.
CASE THIS^.state OF
	stateFlightSimulator.stopped:
		// In STOPPED state:
		// Signal needs to be continuously yellow.
		// Drives needs to be disabled.
		// When enabled go to STARTING state.
		
		// Set signal.
		THIS^.signal.yellow.enable := TRUE;
		
		// Disable drives.
		IF THIS^.isEnabled() THEN
			FOR iCounter := 1 TO 6 BY 1 DO
				Axis[iCounter].enabled := FALSE;
			END_FOR
		END_IF
		
		// If flightsim is enabled go to STARTING state.
		IF THIS^.enabled THEN
			THIS^.state := stateFlightSimulator.starting;
		END_IF
		
	stateFlightSimulator.starting:
		// In STARTING state:
		// Signal needs to be blinking green.
		// Drives needs to be enabled.
		// Once enabled go to neutral position.
		// Once in neutral position go to STARTED state.
	
		// Set signal.
		THIS^.signal.green.enable := TRUE;
		THIS^.signal.green.blink := TRUE;
		
		// Start Axises.
		IF NOT THIS^.isEnabled() THEN
			FOR iCounter := 1 TO 6 BY 1 DO
				Axis[iCounter].enabled := TRUE;
				GVL.servoPositions[iCounter] := 200;
			END_FOR
		END_IF
		
		IF THIS^.isEnabled() AND THIS^.isReady() THEN
			IF NOT bToggle THEN
				// Move pistons to neutral position.
				THIS^.goNeutralPosition();
				bToggle := TRUE;
			ELSE
				// When position has been reached go to started state.
				bToggle := FALSE;
				THIS^.state := stateFlightSimulator.started;
			END_IF	
		END_IF
		
	stateFlightSimulator.started:
		// In STARTED state:
		// Signal needs to be continuously green.
		// When at least one of the drives goes to disabled go to ERROR state.
		// Do movement.
		// When not enabled go to STOPPING state.
	
		// Set signal.
		THIS^.signal.green.enable := TRUE;
		
		// If drives are disabled somehow go to error.
		IF NOT THIS^.isEnabled() THEN
			THIS^.state := stateFlightSimulator.error;
		END_IF
		
		// Do movement.
		THIS^.doMovement(THIS^.newPositions, THIS^.newVelocities);
		
		// If flightsim is disabled go to STOPPING state.
		IF NOT THIS^.enabled THEN
			THIS^.state := stateFlightSimulator.stopping;
		END_IF
		
	stateFlightSimulator.stopping:
		// In STOPPING state:
		// Signal needs to be blinking green.
		// Drives needs to be enabled.
		// Once enabled go to home position.
		// Once in home position go to STOPPED state.
	
		// Set signal.
		THIS^.signal.green.enable := TRUE;
		THIS^.signal.green.blink := TRUE;
		
		// Enable drives if not enabled yet.
		IF NOT THIS^.isEnabled() THEN
			FOR iCounter := 1 TO 6 BY 1 DO
				Axis[iCounter].enabled := TRUE;
			END_FOR
		END_IF
		
		IF THIS^.isEnabled() THEN
			IF NOT bToggle THEN
				// Move pistons to home position.
				THIS^.goHomePosition();
				bToggle := TRUE;
			ELSE
				IF THIS^.isReady() THEN
					// When position has been reached go to stopped state.
					bToggle := FALSE;
					THIS^.state := stateFlightSimulator.stopped;
				END_IF
			END_IF
		END_IF
		
	stateFlightSimulator.error:
		// In ERROR state:
		// Signal needs to be blinking red.
		
		// Set signal.
		THIS^.signal.red.enable := TRUE;
		THIS^.signal.red.blink := TRUE;
		
	stateFlightSimulator.resetting:
		// In RESETTING state:
		// Signal needs to be blinking yellow.
		// If in error drives needs to be reset.
		// Else go to home and go to STOPPED state.
	
		// Set signal.
		THIS^.signal.yellow.enable := TRUE;
		THIS^.signal.yellow.blink := TRUE;
		
		IF THIS^.inError() THEN
			// Reset drives.
			FOR iCounter := 1 TO 6 BY 1 DO
				Axis[iCounter].doReset();
			END_FOR
		ELSE
			// Enable drives if not enabled yet.
			IF NOT THIS^.isEnabled() THEN
				FOR iCounter := 1 TO 6 BY 1 DO
					Axis[iCounter].enabled := TRUE;
				END_FOR
			END_IF
			
			IF THIS^.isEnabled() THEN
				IF NOT bToggle THEN
					// Move pistons to home position.
					THIS^.goHomePosition();
					bToggle := TRUE;
				ELSE
					IF THIS^.isReady() THEN
						// When position has been reached go to stopped state.
						bToggle := FALSE;
						THIS^.state := stateFlightSimulator.stopped;
					END_IF
				END_IF
			END_IF
		END_IF
END_CASE

// Cycle Axis classes.
FOR iCounter := 1 TO 6 BY 1 DO
	THIS^.axis[iCounter].cycle();
END_FOR
// Cycle signal class.
THIS^.signal.cycle();
END_METHOD

METHOD goNeutralPosition : BOOL
VAR
	// Counter to cycle through axis.
	iCounter: INT;
END_VAR
IF THIS^.isReady() THEN
	FOR iCounter := 1 TO 6 BY 1 DO
		THIS^.axis[iCounter].doMovement(position := 200, velocity := 25, continuousUpdate:=FALSE);
	END_FOR
END_IF
END_METHOD

METHOD isReady : BOOL
VAR_INPUT
END_VAR
VAR
	// Counter to cycle through axis.
	iCounter: INT;
END_VAR
// Check ready status of all axis, when one is not ready return with FALSE.
FOR iCounter := 1 TO 6 BY 1 DO
	IF NOT THIS^.axis[iCounter].isReady() THEN
		isReady := FALSE;
		RETURN;
	END_IF;
END_FOR;

isReady := TRUE;
END_METHOD

METHOD doMovement : BOOL
VAR_INPUT
	positions : ARRAY[1..6] OF REAL;
	speeds : ARRAY[1..6] OF REAL;
END_VAR
VAR
	// Counter to cycle through axis.
	iCounter: INT;
	// Var that says its safe to execute this command, will be lowered in the FOR loop check.
	bSafe: BOOL := TRUE;
END_VAR
FOR iCounter := 1 TO 6 BY 1 DO
	// If any of the positions are larger than 390 or smaller than 10 don't execute the command.
	IF positions[iCounter] > 390 OR positions[iCounter] < 10 THEN
		bSafe := FALSE;
	END_IF
	
	// If any of the velocities are larger than 401 or smaller than 0 don't execute the command.
	IF speeds[iCounter] >= 401 OR speeds[iCounter] < 0 THEN
		bSafe := FALSE;
	END_IF
END_FOR

IF bSafe THEN
    FOR iCounter := 1 TO 6 BY 1 DO
        IF positions[iCounter] > 390 THEN
            Axis[iCounter].doMovement(position:=390, velocity:=speeds[iCounter], continuousUpdate:=FALSE);
        ELSIF positions[iCounter] < 10 THEN
            Axis[iCounter].doMovement(position:=100, velocity:=speeds[iCounter], continuousUpdate:=FALSE);
        ELSE
            Axis[iCounter].doMovement(position:=positions[iCounter], velocity:=speeds[iCounter], continuousUpdate:=TRUE);
        END_IF
    END_FOR
END_IF
END_METHOD

METHOD isInitialised : BOOL
VAR_INPUT
END_VAR
VAR
	// Counter to cycle through axis.
	iCounter: INT;
END_VAR
// Check if all axis are initialised, when one is not initialised return with FALSE.
FOR iCounter := 1 TO 6 BY 1 DO
	IF NOT THIS^.axis[iCounter].isInitialised() THEN
		isInitialised := FALSE;
		RETURN;
	END_IF;
END_FOR;

isInitialised := TRUE;
END_METHOD

METHOD init : BOOL
VAR_INPUT
	axis1: REFERENCE TO AXIS_REF_ETC_FESTO_CMMT_AS;
	axis2: REFERENCE TO AXIS_REF_ETC_FESTO_CMMT_AS;
	axis3: REFERENCE TO AXIS_REF_ETC_FESTO_CMMT_AS;
	axis4: REFERENCE TO AXIS_REF_ETC_FESTO_CMMT_AS;
	axis5: REFERENCE TO AXIS_REF_ETC_FESTO_CMMT_AS;
	axis6: REFERENCE TO AXIS_REF_ETC_FESTO_CMMT_AS;
	lightRed: REFERENCE TO BOOL;
	lightYellow: REFERENCE TO BOOL;
	lightGreen: REFERENCE TO BOOL;
	enabled: REFERENCE TO BOOL;
	// When this variable is HIGH it means that the safety system is active.
	// This means none of it's safety systems has been triggered.
	safetySystem: REFERENCE TO BOOL;
	newPositions: REFERENCE TO ARRAY[1..6] OF REAL;
	newVelocities: REFERENCE TO ARRAY[1..6] OF REAL;
END_VAR
THIS^.axis[1].init(axis1);
THIS^.axis[2].init(axis2);
THIS^.axis[3].init(axis3);
THIS^.axis[4].init(axis4);
THIS^.axis[5].init(axis5);
THIS^.axis[6].init(axis6);

THIS^.signal.init(lightRed, lightYellow, lightGreen);

THIS^.enabled REF= enabled;
THIS^.safetySystem REF= safetySystem;

THIS^.newPositions REF= newPositions;
THIS^.newVelocities REF= newVelocities;
END_METHOD

METHOD inError : BOOL
VAR
	// Counter to cycle through axis.
	iCounter: INT;
END_VAR
// Check error status of all axis, when one is in error return with TRUE.
FOR iCounter := 1 TO 6 BY 1 DO
	IF THIS^.axis[iCounter].inError() THEN
		inError := TRUE;
		RETURN;
	END_IF;
END_FOR;

InError := FALSE;
END_METHOD

METHOD goHomePosition : BOOL
VAR
	// Counter to cycle through axis.
	iCounter: INT;
END_VAR
// Abort current movement action.
FOR iCounter := 1 TO 6 BY 1 DO
	THIS^.axis[iCounter].doAbort();
END_FOR

IF THIS^.isReady() THEN
	FOR iCounter := 1 TO 6 BY 1 DO
		THIS^.axis[iCounter].doMovement(position := 10, velocity := 25, continuousUpdate:=FALSE);
	END_FOR
END_IF
END_METHOD

METHOD goTopPosition : BOOL
VAR
	// Counter to cycle through axis.
	iCounter: INT;
END_VAR
// Abort current movement action.
FOR iCounter := 1 TO 6 BY 1 DO
	THIS^.axis[iCounter].doAbort();
END_FOR

IF THIS^.isReady() THEN
	FOR iCounter := 1 TO 6 BY 1 DO
		THIS^.axis[iCounter].doMovement(position := 390, velocity := 25, continuousUpdate:=FALSE);
	END_FOR
END_IF
END_METHOD

END_FUNCTION_BLOCK

// Axis
FUNCTION_BLOCK Axis
VAR
	// Power stage of the servo drive.
	MC_Power: MC_Power;
	// Reset object to reset servo drive.
	MC_Reset: MC_Reset;
	// Move absolute object to move the servo.
	MC_MoveAbsolute: MC_MoveAbsolute;
	// Read object to read current position.
	MC_ReadActualPosition: MC_ReadActualPosition;
	// Read status object to read current status of servo drive.
	MC_ReadStatus: MC_ReadStatus;
	
	// REF to axis.
	axis: REFERENCE TO AXIS_REF_ETC_FESTO_CMMT_AS;
	// Allow move orders to be overwritten by new moveorders.
	continuousUpdate: BOOL := FALSE;
	// Execute a move order.
	execute: BOOL := FALSE;
	// Drive is enabled.
	isEnabled: BOOL := FALSE;
	// Drive is in error.
	error: BOOL := FALSE;
	// Drive is beign reset, toggle bit.
	reset: BOOL := FALSE;
	// Requested position of servo.
	position: REAL := 0;
	// Requested velocity of servo.
	velocity: REAL := 0;
	// Acceleration of servo.
	acceleration: REAL := 5000;
	// Deceleration of servo.
	deceleration: REAL := 5000;
	// Jerk of servo.
	jerk: REAL := 15000;
END_VAR

PROPERTY enabled : BOOL
GET
enabled := THIS^.isEnabled AND (NOT THIS^.MC_ReadStatus.Disabled);
END_GET
SET
THIS^.isEnabled := enabled;
END_SET
END_PROPERTY

METHOD init : BOOL
VAR_INPUT
	axis : REFERENCE TO AXIS_REF_ETC_FESTO_CMMT_AS;
END_VAR
// This function references the servo drive to the instance of the function block.
THIS^.axis REF= axis;
END_METHOD

METHOD doAbort : BOOL
VAR_INPUT
END_VAR
THIS^.execute := FALSE;
END_METHOD

METHOD isReady : BOOL
VAR_INPUT
END_VAR
// Axis is ready when in standstill and not been given an execution order.
isReady := THIS^.MC_ReadStatus.Standstill AND NOT THIS^.execute;
END_METHOD

METHOD doMovement : BOOL
VAR_INPUT
	velocity: REAL := 0;
	position: REAL := 0;
	continuousUpdate: BOOL := FALSE;
END_VAR
// Only do movements when drive is started.
IF THIS^.isEnabled THEN
	THIS^.position := position;
	THIS^.velocity := velocity; 
	THIS^.continuousUpdate := continuousUpdate;
	THIS^.execute := TRUE;
	DoMovement := TRUE;		// return
ELSE
	THIS^.execute := FALSE;
	DoMovement := FALSE;	// return
END_IF;
END_METHOD

METHOD doReset
THIS^.reset := TRUE;
END_METHOD

METHOD getPosition : REAL
VAR_INPUT
END_VAR
IF THIS^.MC_ReadActualPosition.Valid OR (NOT THIS^.MC_ReadActualPosition.Error) THEN
	getPosition := THIS^.MC_ReadActualPosition.Position;
ELSE
	getPosition := -1;
END_IF
END_METHOD

METHOD inError : BOOL
VAR_INPUT
END_VAR
inError := THIS^.error;
END_METHOD


METHOD cycle : BOOL
VAR_INPUT
END_VAR
// Read drive status first
MC_ReadStatus(
	axis := THIS^.axis, 
	Enable := TRUE
);

// Set drive to error if an error occurs.
IF THIS^.MC_ReadStatus.ErrorStop OR THIS^.MC_ReadStatus.Error THEN
	THIS^.error := TRUE;
END_IF

// Function block to enable the drive.
THIS^.MC_Power(
	axis := THIS^.axis,
	Enable := THIS^.isEnabled
);

// Function block to reset the drive.
THIS^.MC_Reset(
	axis := THIS^.axis,
	Execute := THIS^.reset
);

// Reset the reset variable
IF (THIS^.MC_Reset.Done AND THIS^.reset) OR THIS^.MC_Reset.Error THEN
	THIS^.reset := FALSE;
	THIS^.error := FALSE;
END_IF

// Reset execute when movement is done.
IF (THIS^.MC_MoveAbsolute.Done 
//AND NOT THIS^.continuousUpdate
) OR THIS^.MC_MoveAbsolute.CommandAborted OR THIS^.error THEN
	THIS^.execute := FALSE;
END_IF

// Reset the move function if it's in error.
IF NOT THIS^.MC_MoveAbsolute.Error THEN
	// Function block to move the drive.
	THIS^.MC_MoveAbsolute(
		axis := THIS^.axis,
		Execute := THIS^.execute,
		//ContinuousUpdate := THIS^.continuousUpdate,
		position := THIS^.position,
		velocity := THIS^.velocity,
		acceleration := THIS^.acceleration,
		deceleration := THIS^.deceleration,
		jerk := THIS^.jerk
	);
ELSE
	THIS^.MC_MoveAbsolute(axis := THIS^.axis, Execute := FALSE);
END_IF;

// Function block to read the drives current position.
THIS^.MC_ReadActualPosition(
	axis := THIS^.axis,
	Enable := TRUE
);
END_METHOD

METHOD isInitialised : BOOL
VAR_INPUT
END_VAR
isInitialised := THIS^.MC_ReadStatus.Valid;
END_METHOD

END_FUNCTION_BLOCK

// signal
FUNCTION_BLOCK signal
VAR_INPUT
	// Red light.
	red: light;
	// Yellow light.
	yellow: light;
	// Green light.
	green: light;
END_VAR
VAR
	
	// TON.
	clockTON: TON;
	// TOF.
	clockTOF: TOF;
	// Current clock state.
	clock: BOOL;
END_VAR

METHOD init : BOOL
VAR_INPUT
	red: REFERENCE TO BOOL;
	yellow: REFERENCE TO BOOL;
	green: REFERENCE TO BOOL;
END_VAR
VAR
END_VAR
THIS^.red.init(red, clock);
THIS^.yellow.init(yellow, clock);
THIS^.green.init(green, clock);
END_METHOD

METHOD cycle : BOOL
VAR_INPUT
END_VAR
clockTON(IN:= NOT clockTOF.Q, PT:=T#500MS);
clockTOF(IN:= clockTON.Q, PT:=T#500MS);
THIS^.clock := clockTOF.Q;

// Cycle light objects.
THIS^.red.cycle();
THIS^.yellow.cycle();
THIS^.green.cycle();
END_METHOD

END_FUNCTION_BLOCK

// Light
FUNCTION_BLOCK Light
VAR
	light: REFERENCE TO BOOL;
	clock: REFERENCE TO BOOL;
	
	enabled: BOOL := FALSE;
	blinking: BOOL := FALSE;
END_VAR

PROPERTY blink : BOOL
SET
THIS^.blinking := blink;
END_SET
GET
blink := THIS^.blinking;
END_GET
END_PROPERTY

METHOD init : BOOL
VAR_INPUT
	light: REFERENCE TO BOOL;
	clock: REFERENCE TO BOOL;
END_VAR
VAR
END_VAR
THIS^.light REF= light;
THIS^.clock REF= clock;
END_METHOD

METHOD cycle : BOOL
VAR_INPUT
END_VAR
IF THIS^.enabled THEN
	IF THIS^.blinking THEN
		// If blinking is enabled, turn light on or off depending on clock state.
		IF THIS^.clock THEN
			THIS^.light := TRUE;
		ELSE
			THIS^.light := FALSE;
		END_IF
	ELSE
			THIS^.light := TRUE;
	END_IF
ELSE
	THIS^.light := FALSE;
END_IF
END_METHOD

PROPERTY enable : BOOL
GET
enable := THIS^.enabled;
END_GET
SET
THIS^.enabled := enable;
END_SET
END_PROPERTY

END_FUNCTION_BLOCK

// PLC/Application/TcpClient
PROGRAM TcpClient
VAR

    // Client object that connects to client machine.
	fbTcpClient   : NBS.TCP_Client;
    // Read object that reads incomming data from client machine.
	fbTcpRead     : NBS.TCP_Read;
    // Write object that writes data to client machine.
	fbTcpWrite    : NBS.TCP_Write;
	
	// TON object for reset delay.
	tonResetDelay: TON;
	// Received telegram from Read object.
	received      : STRING(gvlSetting.gc_wMaxTelegram);
	// Sent telegram to Write object.
	sent          : STRING(gvlSetting.gc_wMaxTelegram);
	// JSON Parser object to parse read data.
	parseJSON     : JSON_TO_STRUCT;
	// JSON Composer object to compose data to write.
	composeJSON   : STRUCT_TO_JSON;
	// Struct that stores the received data in usable arrays.
	servoData     : ServoData;
    // Make connection.
	xConnect      : BOOL := TRUE;
	// Do composing.
	xCompose: BOOL;
	// Do write action.
	xWrite: BOOL;
	// Do parsing
	xParse: BOOL;
	
	j : INT := 1;
 
    // Do read action.
	xRead         : BOOL;
    // Size of read data telegram.
	udiRead       : UDINT;
	// Timeout in µs.
	udiTimeOut: UDINT := 500000;
	
	
	udiVal        : UDINT;
    pudiVal       : POINTER TO BYTE;
    iIndex        : INT;
	xMissingAck   : BOOL;
    udiResult     : UDINT;
    udiLastAck    : UDINT;
    udiNow        : UDINT;
END_VAR

 fbTcpClient(xEnable := xConnect, ipAddr := gvlSetting.gc_stIpAddr, uiPort := gvlSetting.gc_uiPort, udiTimeOut := udiTimeOut);
// 
// // Run when connection is active.
// IF fbTcpClient.xActive AND GVL.FlightSimulator.isInitialised() THEN
// 	
// 	IF fbTcpWrite.xDone THEN
// 		xWrite := FALSE;
// 	ELSIF NOT fbTcpWrite.xBusy THEN
// 		IF composeJSON.Done AND composeJSON.Execute THEN
// 			xCompose := FALSE;
// 			xWrite := TRUE;
// 		ELSIF (NOT composeJSON.Busy) THEN
// 			   xCompose := TRUE;
// 			   xWrite := FALSE;
// 		END_IF
// 	END_IF
// 	
// 	composeJSON(
// 		Execute:= xCompose,
// 		JSONString:= ADR(sent),
// 		JSONStringSize:= SIZEOF(sent),
// 		JSONVars:= ADR(GVL.currentPositions),
// 		NumberOfVars:= SIZEOF(GVL.currentPositions) / SIZEOF(JSONVAR)
// 	); 
// 	fbTcpWrite(xExecute := xWrite, hConnection := fbTcpClient.hConnection, udiTimeOut := udiTimeOut, szSize := SIZEOF(sent), pData := ADR(sent));
// 	
// 	IF (NOT fbTcpRead.xBusy) AND (NOT parseJSON.Busy) THEN
// 		xRead := TRUE;
// 	ELSIF fbTcpRead.xReady THEN
// 		xRead := FALSE;
// 		xParse := TRUE;
// 	ELSIF (NOT parseJSON.Busy) THEN
// 		xParse := FALSE;
// 	END_IF
// 
// 	parseJSON(
// 		Execute := xParse,
// 		JSONString:= ADR(received),
// 		JSONStringSize:= SIZEOF(received),
// 		JSONVars:= ADR(servoData),
// 		NumberOfVars:= SIZEOF(servoData) / SIZEOF(JSONVAR)
// 	);
// 	
// 	received := '';
// 	//FOR j := 1 TO SIZEOF(received) DO
// 	//	received[j] := 0;
// 	//END_FOR
// 	//sent := '';
// 	fbTcpRead(xEnable := xRead, hConnection := fbTcpClient.hConnection, szSize := SIZEOF(received), pData := ADR(received), szCount => udiRead);
// 	
// END_IF
// 
// // Reset connection when connection has stopped.
// IF (NOT xConnect) THEN
// 	// Reset all variables.
// 	xConnect := FALSE;
// 	xWrite := FALSE;
// 	xCompose := FALSE;
// 	fbTcpWrite(xExecute := FALSE);
// 	xRead := FALSE;
// 	xParse := FALSE;
// 	fbTcpRead(xEnable := FALSE);
// 	received := '';
// 	sent := '';
// 	// Delay reset for 3 sec.
// 	tonResetDelay(IN:=TRUE, PT:=T#3S);
// 	IF (tonResetDelay.Q) THEN
// 		tonResetDelay(IN:=FALSE);
// 		xConnect := TRUE;
// 	END_IF
// 	
// END_IF
// 
// IF fbTcpClient.xDone AND xConnect THEN
// 	xConnect := FALSE;
// END_IF
// 
// // Stop connection when in error.
// //IF fbTcpClient.xError OR fbTcpWrite.xError OR fbTcpRead.xError THEN
// IF fbTcpClient.xError OR fbTcpRead.xError THEN
// 
// 	xConnect := FALSE;
// 	fbTcpWrite(xExecute := FALSE);
// END_IF 
// 

// Run when connection is active.
IF fbTcpClient.xActive AND GVL.FlightSimulator.isInitialised() THEN

    // -------------------------
    //  VERSTUREN NAAR STUARTSERVER
    // -------------------------
    IF fbTcpWrite.xDone THEN
        // Schrijfactie is afgerond → reset write-flag
        xWrite := FALSE;
    ELSIF NOT fbTcpWrite.xBusy THEN
        // Socket is vrij → bouw nieuwe JSON en verstuur

        // Bouw JSON in exact het formaat dat de StuartServer verwacht:
        // {"currentPositions":[p1,p2,p3,p4,p5,p6]}
        sent := '{"currentPositions":[';

        FOR j := 1 TO 6 DO
            // Positie uit GVL.currentPositions (Number-veld)
            sent := CONCAT(sent, REAL_TO_STRING(GVL.currentPositions[j].Number));

            // Komma tussen de waarden, geen komma na de laatste
            IF j < 6 THEN
                sent := CONCAT(sent, ',');
            END_IF
        END_FOR

        // Sluit de JSON af
        sent := CONCAT(sent, ']}');

        // We hebben nu een volledige JSON → start schrijfactie
        xWrite := TRUE;
    END_IF

    // Stuur de inhoud van 'sent' naar de StuartServer
    fbTcpWrite(
        xExecute    := xWrite,
        hConnection := fbTcpClient.hConnection,
        udiTimeOut  := udiTimeOut,
        szSize      := SIZEOF(sent),
        pData       := ADR(sent)
    );

    // -------------------------
    //  ONTVANGEN VAN STUARTSERVER
    // -------------------------
    IF (NOT fbTcpRead.xBusy) AND (NOT parseJSON.Busy) THEN
        xRead := TRUE;
    ELSIF fbTcpRead.xReady THEN
        xRead := FALSE;
        xParse := TRUE;
    ELSIF (NOT parseJSON.Busy) THEN
        xParse := FALSE;
    END_IF

    parseJSON(
        Execute         := xParse,
        JSONString      := ADR(received),
        JSONStringSize  := SIZEOF(received),
        JSONVars        := ADR(servoData),
        NumberOfVars    := SIZEOF(servoData) / SIZEOF(JSONVAR)
    );

    // Buffer leegmaken voor volgende receive
    received := '';
    fbTcpRead(
        xEnable    := xRead,
        hConnection:= fbTcpClient.hConnection,
        szSize     := SIZEOF(received),
        pData      := ADR(received),
        szCount    => udiRead
    );

END_IF


// Reset connection when connection has stopped.
 IF (NOT xConnect) THEN
 	// Reset all variables.
 	xConnect := FALSE;
 	xWrite := FALSE;
 	xCompose := FALSE;
	fbTcpWrite(xExecute := FALSE);
 	xRead := FALSE;
 	xParse := FALSE;
 	fbTcpRead(xEnable := FALSE);
	received := '';
 	sent := '';
 	// Delay reset for 3 sec.
 	tonResetDelay(IN:=TRUE, PT:=T#3S);
 	IF (tonResetDelay.Q) THEN
 		tonResetDelay(IN:=FALSE);
 		xConnect := TRUE;
 	END_IF
	
 END_IF
 
 IF fbTcpClient.xDone AND xConnect THEN
 	xConnect := FALSE;
 END_IF

 // Stop connection when in error.
 //IF fbTcpClient.xError OR fbTcpWrite.xError OR fbTcpRead.xError THEN
IF fbTcpClient.xError OR fbTcpRead.xError THEN

	xConnect := FALSE;
	fbTcpWrite(xExecute := FALSE);
END_IF

END_PROGRAM

// PLC/Application/Main
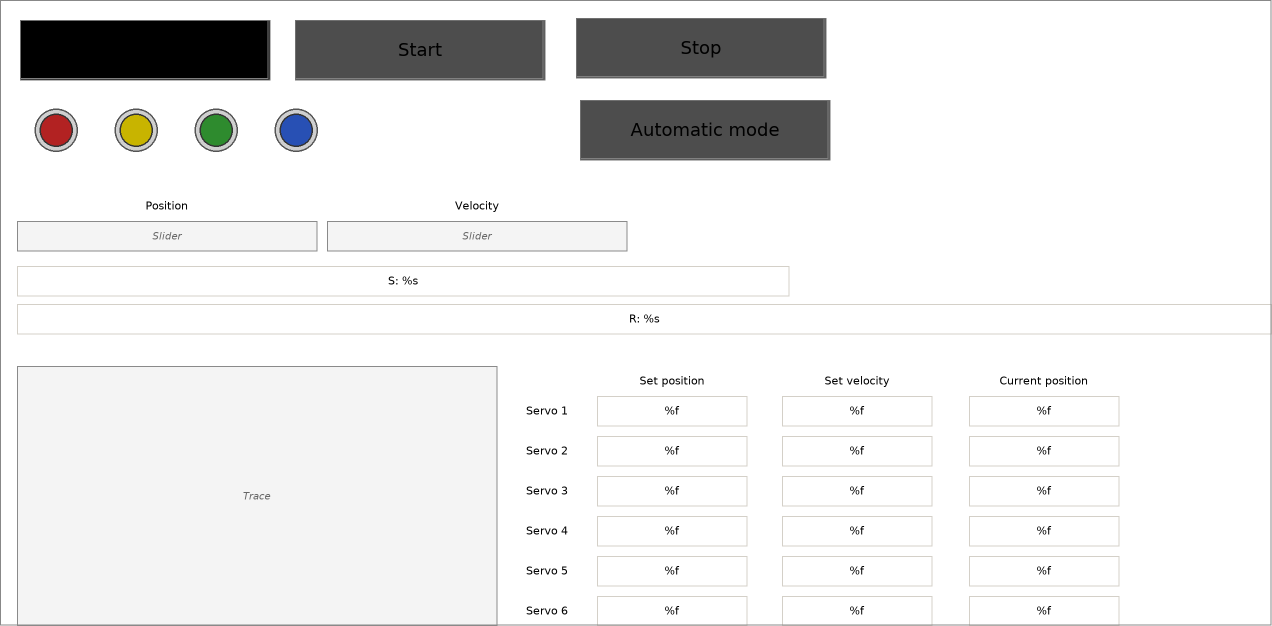
VISUALIZATION Main  // 1272x626
    Button (20,20 250x60), "Reset"
        tap GVL.resetHMI
    Button (295,20 250x60), "Start"
        tap GVL.startHMI
    Slider (17,221 300x30), scale 10..390
    Button (580,100 250x60), "Automatic mode"
        toggle GVL.usetcpdata
    Slider (327,221 300x30), scale 0..400
    Button (576,18 250x60), "Stop"
        tap GVL.stopHMI
    Lamp1 (191,105 50x50), variable: GVL.lightGreen, style: Lamp-Lamp1-Green
    Lamp1 (31,105 50x50), variable: GVL.lightRed, style: Lamp-Lamp1-Red
    Lamp1 (111,105 50x50), variable: GVL.lightYellow, style: Lamp-Lamp1-Yellow
    Textfield (17,266 772x30), "S: %s", text variable: TcpClient.sent
    Textfield (17,304 1255x30), "R: %s", text variable: TcpClient.received
    Textfield (597,396 150x30), "%f", text variable: GVL.servoPositions[1]
        OnMouseClick: write the text variable via InputWithLimits, min 0, max 400
    Textfield (597,436 150x30), "%f", text variable: GVL.servoPositions[2]
        OnMouseClick: write the text variable via InputWithLimits, min 0, max 400
    Textfield (597,476 150x30), "%f", text variable: GVL.servoPositions[3]
        OnMouseClick: write the text variable via InputWithLimits, min 0, max 400
    Textfield (597,516 150x30), "%f", text variable: GVL.servoPositions[4]
        OnMouseClick: write the text variable via InputWithLimits, min 0, max 400
    Textfield (597,556 150x30), "%f", text variable: GVL.servoPositions[5]
        OnMouseClick: write the text variable via InputWithLimits, min 0, max 400
    Textfield (597,596 150x30), "%f", text variable: GVL.servoPositions[6]
        OnMouseClick: write the text variable via InputWithLimits, min 0, max 400
    Textfield (782,396 150x30), "%f", text variable: GVL.servoVelocities[1]
        OnMouseClick: write the text variable via InputWithLimits, min 0, max 400
    Textfield (782,436 150x30), "%f", text variable: GVL.servoVelocities[2]
        OnMouseClick: write the text variable via InputWithLimits, min 0, max 400
    Textfield (782,476 150x30), "%f", text variable: GVL.servoVelocities[3]
        OnMouseClick: write the text variable via InputWithLimits, min 0, max 400
    Textfield (782,516 150x30), "%f", text variable: GVL.servoVelocities[4]
        OnMouseClick: write the text variable via InputWithLimits, min 0, max 400
    Textfield (782,556 150x30), "%f", text variable: GVL.servoVelocities[5]
        OnMouseClick: write the text variable via InputWithLimits, min 0, max 400
    Textfield (782,596 150x30), "%f", text variable: GVL.servoVelocities[6]
        OnMouseClick: write the text variable via InputWithLimits, min 0, max 400
    Label (597,366 150x30), "Set position"
    Label (782,366 150x30), "Set velocity"
    Label (497,396 100x30), "Servo 1"
    Label (497,436 100x30), "Servo 2"
    Label (497,476 100x30), "Servo 3"
    Label (497,516 100x30), "Servo 4"
    Label (497,556 100x30), "Servo 5"
    Label (497,596 100x30), "Servo 6"
    Lamp1 (271,105 50x50), variable: GVL.FlightSimulator.isReady(), style: Lamp-Lamp1-Blue
    Trace (17,366 480x260)
    Textfield (969,396 150x30), "%f", text variable: GVL.servoPositionsCurrent[1]
        OnMouseClick: write the text variable via InputWithLimits, min 0, max 400
    Textfield (969,436 150x30), "%f", text variable: GVL.servoPositionsCurrent[2]
        OnMouseClick: write the text variable via InputWithLimits, min 0, max 400
    Textfield (969,476 150x30), "%f", text variable: GVL.servoPositionsCurrent[3]
        OnMouseClick: write the text variable via InputWithLimits, min 0, max 400
    Textfield (969,516 150x30), "%f", text variable: GVL.servoPositionsCurrent[4]
        OnMouseClick: write the text variable via InputWithLimits, min 0, max 400
    Textfield (969,556 150x30), "%f", text variable: GVL.servoPositionsCurrent[5]
        OnMouseClick: write the text variable via InputWithLimits, min 0, max 400
    Textfield (969,596 150x30), "%f", text variable: GVL.servoPositionsCurrent[6]
        OnMouseClick: write the text variable via InputWithLimits, min 0, max 400
    Label (969,366 150x30), "Current position"
    Label (92,191 150x30), "Position"
    Label (402,191 150x30), "Velocity"
END_VISUALIZATION
